{attribute 'qualified_only'}
{attribute 'strict'}
{attribute 'to_string'}
TYPE E_ServoliftCommand :
(
	Idle := 0,  // De servolift geen actie laten uitvoeren
	Beweegomhoog, // De servolift omhoog bewegen
	Beweegomlaag, // De servolift omlaag bewegen
	Houdtvast // De servolift zijn positie laten vasthouden
);
END_TYPE

(* stored: Version 1.1.0.1
   DUT E_ServoliftCommand: Id {83e0a771-ea57-4521-99e1-c509e6b4a008} *)
